// TIA Portal V18 export
TYPE "ProcessDatad"
   STRUCT
      PartStatus : Int;   // 产品状态 / PartStatus
      PartSNGCode : Int;   // 产品NG代码 / PartSNGCode
      PartRemoveFlag : Bool;   // PartRemoveFlag
      Spare1 : Bool;   // Spare1
      Spare2 : Bool;   // Spare2
      Spare3 : Bool;   // Spare3
      Spare4 : Bool;   // Spare4
      Spare5 : Bool;   // Spare5
      Spare6 : Bool;   // Spare6
      Spare7 : Bool;   // Spare7
      Spare8 : Bool;   // Spare8
      Spare9 : Bool;   // Spare9
      Spare10 : Bool;   // Spare10
      Spare11 : Bool;   // Spare11
      Spare12 : Bool;   // Spare12
      Spare13 : Bool;   // Spare13
      Spare14 : Bool;   // Spare14
      Spare15 : Bool;   // Spare15
      ShaftCode { S7_SetPoint := 'True'} : String[128];   // 轴条码 / ShaftCode
      RingCode_1 { S7_SetPoint := 'True'} : String[128];   // 条码 / RingCode_1
      Code_1 : String[128];   // Code_1
      RingCode_2 : String[128];   // RingCode_2
      TableCode_1 : String[128];   // TableCode_1
      TableCode_2 : String[128];   // TableCode_2
      Press1Program : Int;   // Press1Program
      Press1FinalPosition : Real;   // Press1FinalPosition
      Press1FinalForce : Real;   // Press1FinalForce
      Press2Program : Int;   // Press2Program
      Press2FinalPosition : Real;   // Press2FinalPosition
      Press2FinalForce : Real;   // Press2FinalForce
      IV3_ShaftCheckResult : Int;   // IV3_ShaftCheckResult
      IV3_ShaftScore_1 : Int;   // IV3_ShaftScore_1
      IV3_ShaftScore_2 : Int;   // IV3_ShaftScore_2
      IV3_ShaftScore_3 : Int;   // IV3_ShaftScore_3
      IV3_ShaftScore_4 : Int;   // IV3_ShaftScore_4
      IV3_MagnetCheckResult : Int;   // IV3_MagnetCheckResult
      IV3_MagnetScore : Int;   // IV3_MagnetScore
      IV3_ShaftScoreTotal : Real;   // IV3_ShaftScore_4
      Spare_3 : Array[0..88] of Int;
   END_STRUCT;
END_TYPE
